// TIA Portal V19 export
DATA_BLOCK "InstCallGlobal"   // DB25
// stored: InstanceOfName CallGlobal, InstanceOfType FB
"CallGlobal"
   // VAR
   //    statClockSysMemOld { ExternalWritable := 'False'} : Byte;
   //    instLAF_PowerOnOff { ExternalWritable := 'False'} : "LAF_PowerOnOff";
   //    instLAF_HmiHeaderManager { ExternalWritable := 'False'} : "LAF_HmiHeaderManager";
   //    instLAF_ClockGen { ExternalWritable := 'False'} : "LAF_ClockGenerator";
   //    instLSNTP_Server { ExternalWritable := 'False'} : "LSNTP_Server";
   // END_VAR
BEGIN
END_DATA_BLOCK
